//Index0x7000   Subindex 16#3
TYPE
    Iv3InputRequestResponse3 :
    STRUCT
        Bit0                     : BIT;
        SwitchProgrammNumberBit1 : BIT;
        Bit2                     : BIT;
        Bit3                     : BIT;
        Bit4                     : BIT;
        Bit5                     : BIT;
        Bit6                     : BIT;
        Bit7                     : BIT;
        Bit8                     : BIT;
        Bit9                     : BIT;
        Bit10                    : BIT;
        Bit11                    : BIT;
        Bit12                    : BIT;
        Bit13                    : BIT;
        Bit14                    : BIT;
        Bit15                    : BIT;

    END_STRUCT
END_TYPE

(* stored: Version 1.1.0.1, ProductVersion 3.1.4024.12
   DUT Iv3InputRequestResponse3: Id {f2f2a219-40d3-04a6-0806-a568a5dbe73d} *)
